Fanuc KAREL source: kt00554.KL

-- PROVISIONAL review KL for V770-1; original PC SHA256 eae379aa6dbcabb525ff2e3b7df3699d278ecc6a5e4bd8a33bb1e503d7c73bce
-- Incomplete behavior may be omitted. Consult companion uncertainty JSON. Do not deploy.
PROGRAM KT00554
%NOLOCKGROUP
-- UNRESOLVED_DECL V1 type=000013
-- UNRESOLVED_DECL V2 type=000013
-- UNRESOLVED_DECL OUT type=000013
BEGIN
  -- UNRESOLVED_PC offsets 5-20; opcodes 2E,22,32,35
  -- UNRESOLVED_PC offsets 25-40; opcodes 2E,22,32,35
  -- UNRESOLVED_PC offsets 45-60; opcodes 2E,22,32,35
  -- UNRESOLVED_PC offsets 65-80; opcodes 2E,22,32,35
  -- UNRESOLVED_PC offsets 85-109; opcodes 49,49,92,4A
  -- UNRESOLVED_PC offsets 114-118; opcodes 7F
END KT00554
